KUKA KRL program: LAB_PATHS.src, LAB_PATHS.dat

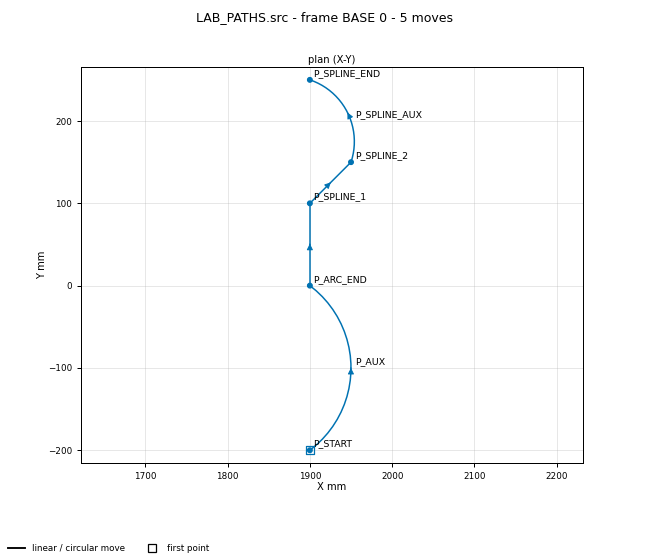
[picture p0: tool path of LAB_PATHS.src in frame BASE 0, 5 of 6 moves have a stored position in this frame; points joined in program order, loops and branches not executed]
--- LAB_PATHS.src ---
&ACCESS RVP
&REL 1
&PARAM TEMPLATE = C:\KRC\Roboter\Template\vorgabe
&PARAM EDITMASK = *
DEF LAB_PATHS()
  ; KLAB fixture: synthetic virtual-only CIRC + CP SPLINE seed
  BAS(#INITMOV,0)
  $ADVANCE=3
  $IPO_MODE=#BASE
  $ORI_TYPE=#VAR
  BAS(#TOOL,0)
  BAS(#BASE,0)
  $ACC.CP=1.0
  $VEL.ORI1=100
  $VEL.ORI2=100
  $ACC.ORI1=100
  $ACC.ORI2=100
  $APO.CDIS=0
  $APO.CPTP=0
  BAS(#VEL_PTP,20)
  BAS(#ACC_PTP,20)
  PTP A_HOME
  PTP P_START
  $VEL.CP=0.1
  CIRC P_AUX,P_ARC_END
  SPLINE
    SLIN P_SPLINE_1
    SPL P_SPLINE_2
    SCIRC P_SPLINE_AUX,P_SPLINE_END
  ENDSPLINE
END

--- LAB_PATHS.dat ---
&ACCESS RVP
&REL 1
DEFDAT LAB_PATHS PUBLIC
  DECL E6AXIS A_HOME={A1 0,A2 -90,A3 90,A4 0,A5 0,A6 0,E1 0,E2 0,E3 0,E4 0,E5 0,E6 0}
  DECL E6POS P_START={X 1900,Y -200,Z 1200,A 180,B 0,C 180,S 2,T 2,E1 0,E2 0,E3 0,E4 0,E5 0,E6 0}
  DECL E6POS P_AUX={X 1950,Y -100,Z 1200,A 180,B 0,C 180,S 2,T 2,E1 0,E2 0,E3 0,E4 0,E5 0,E6 0}
  DECL E6POS P_ARC_END={X 1900,Y 0,Z 1200,A 180,B 0,C 180,S 2,T 2,E1 0,E2 0,E3 0,E4 0,E5 0,E6 0}
  DECL E6POS P_SPLINE_1={X 1900,Y 100,Z 1200,A 180,B 0,C 180,S 2,T 2,E1 0,E2 0,E3 0,E4 0,E5 0,E6 0}
  DECL E6POS P_SPLINE_2={X 1950,Y 150,Z 1200,A 180,B 0,C 180,S 2,T 2,E1 0,E2 0,E3 0,E4 0,E5 0,E6 0}
  DECL E6POS P_SPLINE_AUX={X 1950,Y 200,Z 1200,A 180,B 0,C 180,S 2,T 2,E1 0,E2 0,E3 0,E4 0,E5 0,E6 0}
  DECL E6POS P_SPLINE_END={X 1900,Y 250,Z 1200,A 180,B 0,C 180,S 2,T 2,E1 0,E2 0,E3 0,E4 0,E5 0,E6 0}
ENDDAT
